(* CODESYS project PID_controller.project

Project tree, tasks and I/O mapping:
  Device : CODESYS Control Win V3, 3S - Smart Software Solutions GmbH, order no. 305021, version 3.5.4.10
    application Application
      libraries: Standard, * (System)
      task MainTask (cyclic, interval t#20ms, priority 1) calls Test_PID_Heat2
      task VISU_TASK (cyclic, interval 100 ms, priority 31) calls VisuElems.Visu_Prg
      global variables GVL_Input
      global variables GVL_Output
      global variables GVL_Memory
      global variables GVL_Data
      PID/
        function block PID_controller [ST]
      trace HeatTrace (task MainTask): Test_PID_Heat2.HeatExchanger2_0.Heat_In, Test_PID_Heat2.SP, Test_PID_Heat2.HeatExchanger2_0.Temp
      Progs/
        program Test_PID_Heat2 [LD]
        program Test_PID_Heatx [LD]
        program Test_PID [LD]
      visualisation Tanken
      trace TankTrace (task MainTask): Test_PID.RedBull.Level, Test_PID.PID_0.SP
      Models/
        function block Tank [ST]
        function block HeatExchanger [ST]
        function block HeatExchanger2 [ST]
      visualisation House
  text list GlobalTextList
*)

// Device/Application/GVL_Input
VAR_GLOBAL
	Knapp1: BOOL; // Knapp på våning 1
	Knapp2: BOOL; // 
	Knapp3: BOOL;
	Knapp4: BOOL;
	Vaning1 :BOOL;
	Vaning2 :BOOL;
	Vaning3 :BOOL;
	Vaning4 :BOOL;
	Manuell :BOOL;
	Auto :BOOL;
	Upp :BOOL;
	Ner  :BOOL;
	Service_reset :BOOL;
END_VAR

// Device/Application/GVL_Output
VAR_GLOBAL
	Lampa1 :BOOL;
	Lampa2 :BOOL;
	Lampa3 :BOOL;
	Lampa4 :BOOL;
	HissUpp :BOOL;
	HissNer :BOOL;
	HissDorr :BOOL;
	LampaAuto :BOOL;
	
END_VAR

// Device/Application/GVL_Memory
VAR_GLOBAL
END_VAR

// Device/Application/GVL_Data
VAR_GLOBAL
END_VAR

// Device/Application/Progs/Test_PID_Heat2
PROGRAM Test_PID_Heat2
VAR
	PID_controller_0: PID_controller;
	HeatExchanger2_0: HeatExchanger2;
	SP: REAL := 300;
	Temp_out: REAL := 270;
END_VAR

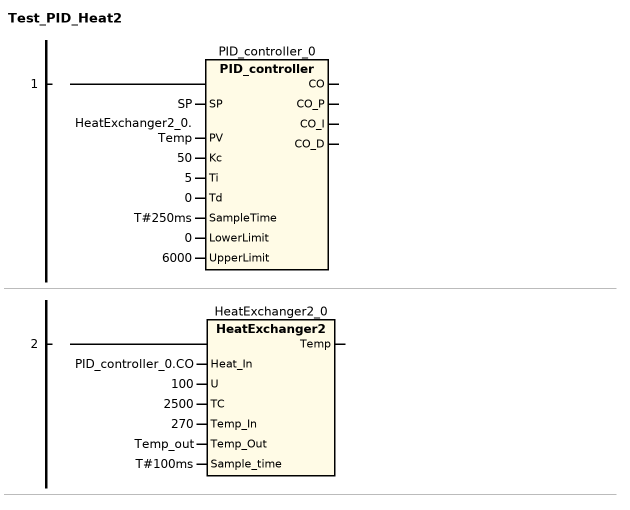
// NETWORK 1
//   HeatExchanger2_0.Temp: The resulting room temperature
PID_controller_0(
    SP := SP,
    PV := HeatExchanger2_0.Temp,
    Kc := 50,
    Ti := 5,
    Td := 0,
    SampleTime := T#250ms,
    LowerLimit := 0,
    UpperLimit := 6000); // PID_controller

// NETWORK 2
//   PID_controller_0.CO: Controller Output
HeatExchanger2_0(
    Heat_In := PID_controller_0.CO,
    U := 100,
    TC := 2500,
    Temp_In := 270,
    Temp_Out := Temp_out,
    Sample_time := T#100ms); // HeatExchanger2

END_PROGRAM

// Device/Application/PID/PID_controller
//***************************************************************
//* A simple PID controller for Codesys.
//* by Alexander Jaworowski
//* Inspiration from https://github.com/br3ttb/Arduino-PID-Library
//* https://github.com/alexjaw/PID_controller
//* This Library is licensed under a MIT License
//
// 2015-02-22	Bug fix in the calculation of CO_I.
//				Added derivative term (d(err)/dt = -d(PV)/dt, i.e.
//				derivative on measurements
//***************************************************************
FUNCTION_BLOCK PID_controller
VAR_INPUT
	SP : REAL;
	PV : REAL;
	Kc : REAL;
	Ti : REAL;
	Td : REAL;
	SampleTime: TIME; //Should be ~0.1 * Tp, Tp : the process time [http://www.controlguru.com/2007/012807.html]
	LowerLimit: REAL;
	UpperLimit: REAL;
END_VAR
VAR_OUTPUT
	CO: REAL; //Controller Output
	CO_P: REAL; //Prportional term
	CO_I: REAL; //Integral term
	CO_D: REAL; //Derivative term
END_VAR
VAR CONSTANT
	millis: UINT := 1000;
END_VAR
VAR
	now: TIME := T#0S;
	lastTime: TIME := T#0S;
	err: REAL := 0; //Process error
	lastCO_P: REAL := 0;  //Used for calculation of the derivative term
	delta_t: REAL;
	lastPV: REAL := 0;
END_VAR

//Check parameters
//Ti division by zero
IF Ti = 0 THEN
	Ti := 1;
END_IF

//Update PID parameters every sampleTime
now := TIME();
IF ((now - lastTime) > SampleTime) THEN
	err := SP - PV;
	delta_t := TIME_TO_REAL(SampleTime)/millis;
	CO_P := Kc * err;
	CO_I := CO_I + 1/Ti * CO_P * delta_t;
	//Add wind-up for CO_I
	IF CO_I < LowerLimit THEN
		CO_I := LowerLimit;
	ELSIF CO_I > UpperLimit THEN
		CO_I := UpperLimit;
	END_IF;
	
	//Observe that d(err)/dt = d(SP)/dt - d(PV)/dt
	//If SP constant,
	//d(err)/dt = - d(PV)/dt
	//Good: no output spikes
	//Bad: some processes need more aggressive tuning
	IF delta_t <> 0 THEN
		CO_D := Td * (PV - lastPV)/delta_t;
	END_IF;
	
	//A different approch would be with a tunable filter
	
	CO := CO_P + CO_I + CO_D;
	//Add wind-up for CO
	IF CO < LowerLimit THEN
		CO := LowerLimit;
	ELSIF CO > UpperLimit THEN
		CO := UpperLimit;
	END_IF;
	
	lastTime := now;
	lastPV := PV;
END_IF;

END_FUNCTION_BLOCK

// Device/Application/Models/HeatExchanger2
// AJ Jaworowski 2015-02-23
// Following the presentation on
// http://openenergymonitor.org/emon/node/2999
FUNCTION_BLOCK HeatExchanger2
VAR_INPUT
	Heat_In:		REAL;		//In principle a radiator in the room [W]
	U:				REAL;		//Thermal conductance [W/K]
	TC:				REAL;		//Thermal capacity [J/K], commonly cv, specific heat capacity [J/kgK]
								//we use a smaller value than in reality, so that we can see changes
								//during a life-time...
	Temp_In:		REAL;		//Start temperature in the room [K]
	Temp_Out:		REAL;		//Outside temperature [K] 
	Sample_time:	TIME;
END_VAR
VAR_OUTPUT
	Temp:			REAL;		//The resulting room temperature
END_VAR
VAR
	now: TIME;
	lastTime: TIME := T#0s;
	delta_t: REAL;
	heat_flow: REAL;
	lastTemp: REAL;
END_VAR
VAR CONSTANT
	millis: REAL := 1000;
END_VAR

now := TIME();
IF ((now - lastTime) > Sample_time) THEN
	delta_t := TIME_TO_REAL(Sample_time)/millis;
	
	//First calculate net heat
	//Heat_In is our heat source
	//Second term is heat flow depending on temperature difference
	//Obs: At start, set lastTime to start temp Temp_In
	IF lastTime = T#0S THEN
		lastTemp := Temp_In;
	END_IF
	heat_flow := Heat_In - U * (lastTemp - Temp_Out);
	
	//Second: calculate temperature change due to heat_flow
	Temp := lastTemp + heat_flow * delta_t / TC;
	
	//Update variables for next iteration
	lastTemp := Temp;
	lastTime := now;
END_IF;

END_FUNCTION_BLOCK

// Device/Application/Progs/Test_PID_Heatx
PROGRAM Test_PID_Heatx
VAR
	PID_0: PID_controller;
	Process_out: REAL := 100;
	SetPoint: REAL := 20;
	A_room_with_a_view: HeatExchanger;
END_VAR

VAR CONSTANT
END_VAR

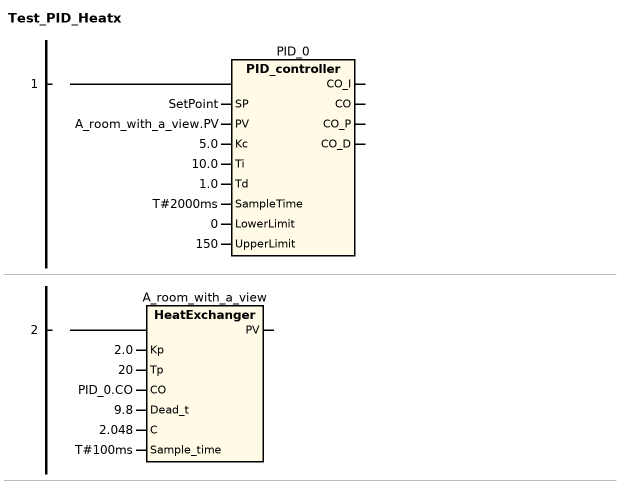
// NETWORK 1
//   A_room_with_a_view.PV: Process value at t1
PID_0(
    SP := SetPoint,
    PV := A_room_with_a_view.PV,
    Kc := 5.0,
    Ti := 10.0,
    Td := 1.0,
    SampleTime := T#2000ms,
    LowerLimit := 0,
    UpperLimit := 150); // PID_controller

// NETWORK 2
//   PID_0.CO: Controller Output
A_room_with_a_view(Kp := 2.0, Tp := 20, CO := PID_0.CO, Dead_t := 9.8, C := 2.048, Sample_time := T#100ms); // HeatExchanger

END_PROGRAM

// Device/Application/Models/HeatExchanger
// AJ Jaworowski 2015-02-22
// Following the recipe by  Peter Nachtwey
// http://www.controlguru.com/wp/p80.html
FUNCTION_BLOCK HeatExchanger
VAR_INPUT
	Kp: REAL; //System gain
	Tp: REAL; //Process time
	CO: REAL; //Output from controller
	Dead_t: REAL; //The time before the system responds to the disturbance
	C: REAL; //Initial steady state value
	Sample_time: TIME;
END_VAR
VAR_OUTPUT
	PV: REAL; //Process value at t1
END_VAR
VAR
	now: TIME;
	lastTime: TIME;
	lastPV:REAL := 140;
	A: REAL;
	B: REAL;
	delta_t: REAL;
END_VAR
VAR CONSTANT
	millis: REAL := 1000;
END_VAR

now := TIME();
IF ((now - lastTime) > Sample_time) THEN
	delta_t := TIME_TO_REAL(Sample_time)/millis;
	A := EXP(-delta_t/Tp);
	B := 1 - A;
	C := 2;
	
	//PV := A * lastPV + B * Kp * CO + C;
	PV := 0.987 * lastPV - 0.00679 * CO + C;
	lastPV := PV;

	lastTime := now;
END_IF

END_FUNCTION_BLOCK

// Device/Application/Models/Tank
//A.J. Jaworowski 2015-02-20
//Simulering av en tank med RedBull
FUNCTION_BLOCK Tank
VAR_INPUT
	Process_In: REAL;  //Flöde in per sekund, testa vad som händer on du matar in 100
					   //Därefter ska regulatorns OUT in i denna ingång.
	Process_Out: REAL; //Flöde ut per sekund, typ 90
					   //Effekten blir att tanken fylls med 10 per sekund
					   //Full efter ca 1 minut - testa
	SampleTime: TIME;  //Uppdateringstid, typ 100ms
	Lower_limit: REAL; //Tankens lägsta nivå, typ 0
	Upper_limit: REAL; //Tankens max nivå, kanske 500
END_VAR
VAR_OUTPUT
	Level: REAL; //Nivån i tanken
END_VAR
VAR
	now: TIME;
	lastTime: TIME;
	proc_sum_in: REAL := 0;
	proc_sum_out: REAL := 0;
	temp: REAL;
	millis: UINT := 1000;
	proc_out: REAL;
END_VAR

now := TIME();
IF ((now - lastTime) > SampleTime) THEN
	Level := Level +  TIME_TO_REAL(SampleTime)/millis * (Process_In - Process_Out);
	IF Level < Lower_limit THEN
		Level := Lower_limit;
	ELSIF Level > Upper_limit THEN
		Level := Upper_limit;
	END_IF;
	lastTime := now;
END_IF;

END_FUNCTION_BLOCK

// Device/Application/Progs/Test_PID
PROGRAM Test_PID
VAR
	PID_0: PID_controller;
	RedBull: Tank;
	Process_out: REAL := 100;
	SetPoint: REAL := 250;
END_VAR

VAR CONSTANT
END_VAR

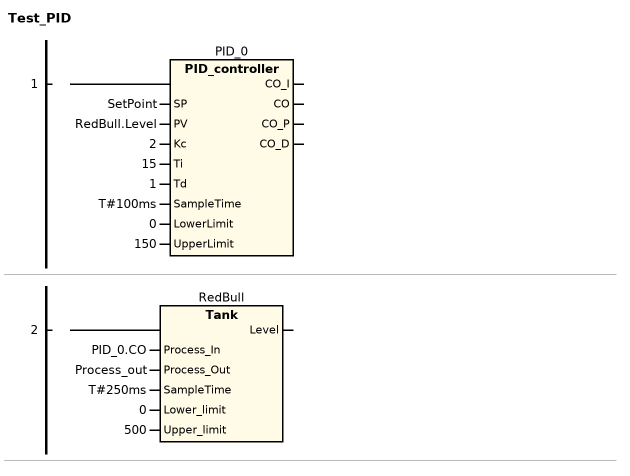
// NETWORK 1
//   RedBull.Level: Nivån i tanken
PID_0(
    SP := SetPoint,
    PV := RedBull.Level,
    Kc := 2,
    Ti := 15,
    Td := 1,
    SampleTime := T#100ms,
    LowerLimit := 0,
    UpperLimit := 150); // PID_controller

// NETWORK 2
//   PID_0.CO: Controller Output
RedBull(
    Process_In := PID_0.CO,
    Process_Out := Process_out,
    SampleTime := T#250ms,
    Lower_limit := 0,
    Upper_limit := 500); // Tank

END_PROGRAM

// Device/Application/Tanken
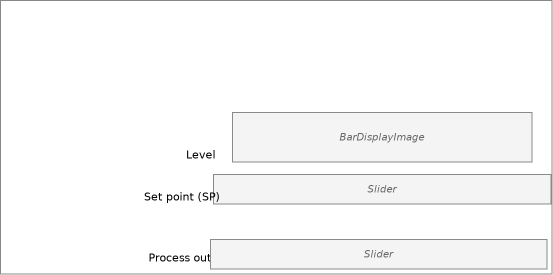
VISUALIZATION Tanken  // 553x275
    BarDisplayImage (232,112 300x50), value: Test_PID.RedBull.Level, style: BarDisplayImage-Gray, scale format: %.1f, scale 0..500
    Label (126,140 150x30), "Level"
    Label (105,243 150x30), "Process out"
    Slider (213,174 338x30), variable: Test_PID_Heatx.SetPoint, scale 0..500
    Label (107,182 150x30), "Set point (SP)"
    Slider (210,239 337x30), variable: Test_PID_Heatx.Process_out, scale 0..300
END_VISUALIZATION

// Device/Application/House
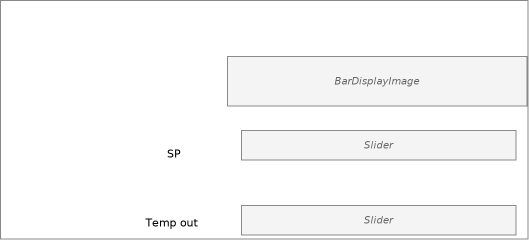
VISUALIZATION House  // 529x240
    BarDisplayImage (227,56 300x50), value: Test_PID_Heat2.HeatExchanger2_0.Temp, style: BarDisplayImage-Gray, scale format: %.1f, scale 270..310
    Slider (241,130 275x30), variable: Test_PID_Heat2.SP, scale 270..310
    Label (99,139 150x30), "SP"
    Slider (241,205 275x30), variable: Test_PID_Heat2.Temp_out, scale 270..310
    Label (97,208 150x30), "Temp out"
END_VISUALIZATION
